// Mitsubishi GX Works2 project: 프로틴 음료 제조기 레더도   PLC: Q00J

PROGRAM MAIN
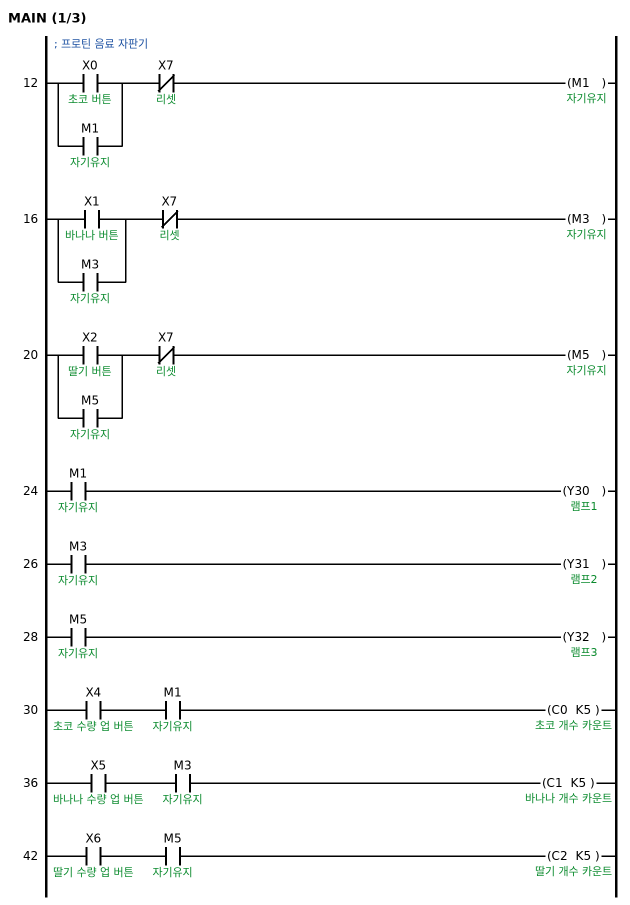
; 프로틴 음료 자판기
12    LD      X0  ; 초코 버튼
      OR      M1  ; 자기유지
      ANI     X7  ; 리셋
      OUT     M1  ; 자기유지
16    LD      X1  ; 바나나 버튼
      OR      M3  ; 자기유지
      ANI     X7  ; 리셋
      OUT     M3  ; 자기유지
20    LD      X2  ; 딸기 버튼
      OR      M5  ; 자기유지
      ANI     X7  ; 리셋
      OUT     M5  ; 자기유지
24    LD      M1  ; 자기유지
      OUT     Y30  ; 램프1
26    LD      M3  ; 자기유지
      OUT     Y31  ; 램프2
28    LD      M5  ; 자기유지
      OUT     Y32  ; 램프3
30    LD      X4  ; 초코 수량 업 버튼
      AND     M1  ; 자기유지
      OUT     C0 K5  ; 초코 개수 카운트
36    LD      X5  ; 바나나 수량 업 버튼
      AND     M3  ; 자기유지
      OUT     C1 K5  ; 바나나 개수 카운트
42    LD      X6  ; 딸기 수량 업 버튼
      AND     M5  ; 자기유지
      OUT     C2 K5  ; 딸기 개수 카운트
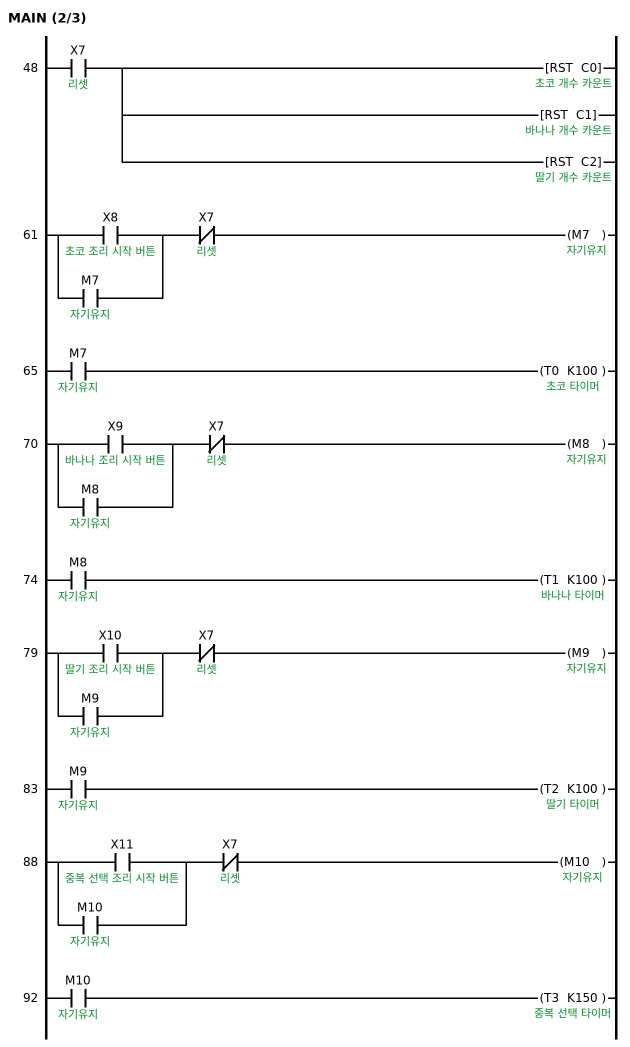
48    LD      X7  ; 리셋
      RST     C0  ; 초코 개수 카운트
      RST     C1  ; 바나나 개수 카운트
      RST     C2  ; 딸기 개수 카운트
61    LD      X8  ; 초코 조리 시작 버튼
      OR      M7  ; 자기유지
      ANI     X7  ; 리셋
      OUT     M7  ; 자기유지
65    LD      M7  ; 자기유지
      OUT     T0 K100  ; 초코 타이머
70    LD      X9  ; 바나나 조리 시작 버튼
      OR      M8  ; 자기유지
      ANI     X7  ; 리셋
      OUT     M8  ; 자기유지
74    LD      M8  ; 자기유지
      OUT     T1 K100  ; 바나나 타이머
79    LD      X10  ; 딸기 조리 시작 버튼
      OR      M9  ; 자기유지
      ANI     X7  ; 리셋
      OUT     M9  ; 자기유지
83    LD      M9  ; 자기유지
      OUT     T2 K100  ; 딸기 타이머
88    LD      X11  ; 중복 선택 조리 시작 버튼
      OR      M10  ; 자기유지
      ANI     X7  ; 리셋
      OUT     M10  ; 자기유지
92    LD      M10  ; 자기유지
      OUT     T3 K150  ; 중복 선택 타이머
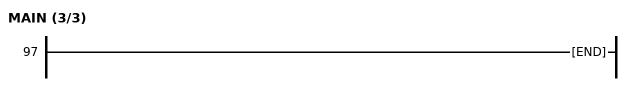
97    END
END_PROGRAM
